Staubli VAL3: IO.pjx

Parameters version=s7.3 stackSize=5000 millimeterUnit=true
Program file=init.pgx
Program file=readme.pgx
Program file=speedCase0_15.pgx
Program file=tableSpeed.pgx
Data file=IO.dtx
